TYPE stFrame :
STRUCT
	frameId: UINT;
END_STRUCT
END_TYPE

(* stored: Version 1.1.0.1, ProductVersion 3.1.4026.18
   DUT stFrame: Id {29c010b8-628c-4280-b317-dd01751f0622} *)
